TYPE ST_LaudaReadCommands_Temperature :
STRUCT
	TemperatureSetpoint					: STRING := 'IN_SP_00';
	BathTemperatureOutflow_01C			: STRING := 'IN_PV_00';
	BathTemperatureOutflow_001C			: STRING := 'IN_PV_10';
	QueryControlledTemperature			: STRING := 'IN_PV_01';
	ExternalTemperature_Pt_C			: STRING := 'IN_PV_03';
	ExternalTemperature_AnalogInput		: STRING := 'IN_PV_04';
	ExternalTemperature_Pt_001_C		: STRING := 'IN_PV_13';
	OvertemperatureTurnoffPoint_Tmax	: STRING := 'IN_SP_03';
	OutflowLimmitHigh					: STRING := 'IN_SP_04';
	OutflowLimmitLow					: STRING := 'IN_SP_05';
	SafetyModeTemperature 				: STRING := 'IN_SP_07';
END_STRUCT
END_TYPE

(* stored: Version 1.1.0.1, ProductVersion 3.1.4024.12
   DUT ST_LaudaReadCommands_Temperature: Id {511096ae-aa9b-4720-bc35-8a5e626e642f} *)
